TYPE ConfigManagerProcesses :
STRUCT
	///Save the currently active config to disk
	save: WriteXmlProcess;
	///Load the config from disk
	load: ReadXmlProcess;
	///Activate the loaded config
	activate: ActivateProcess;
END_STRUCT
END_TYPE

(* stored: Version 1.1.0.1, ProductVersion 3.1.4019.2
   DUT ConfigManagerProcesses: Id {b3504d77-dbc2-49ba-bb1c-6b4fee55374a} *)
